# EPICS StreamDevice protocol: protocols/continuous.proto
Terminator = CR;
ExtraInput = Ignore;

getContinuousStatus {
	in "%39c";
}
